PROGRAM main
VAR
	MainGreen : bool := True;
	MainYellow : bool := False;
	MainRed : bool := False;
	SideGreen : bool := False;
	SideYellow : bool := False;
	SideRed : bool := True;
	CarWaiting : bool := False;
	PedWaiting : bool := False;
	GreenTimer : TON;
	YellowTimer : TON;
	SideGreenTimer : TON;
	SideYellowTimer : TON;
	SideYeIIowTimer : dint;
	CycIeActive : bool := False;
	CycleActive : bool := False;
	TON0 : TON;
END_VAR

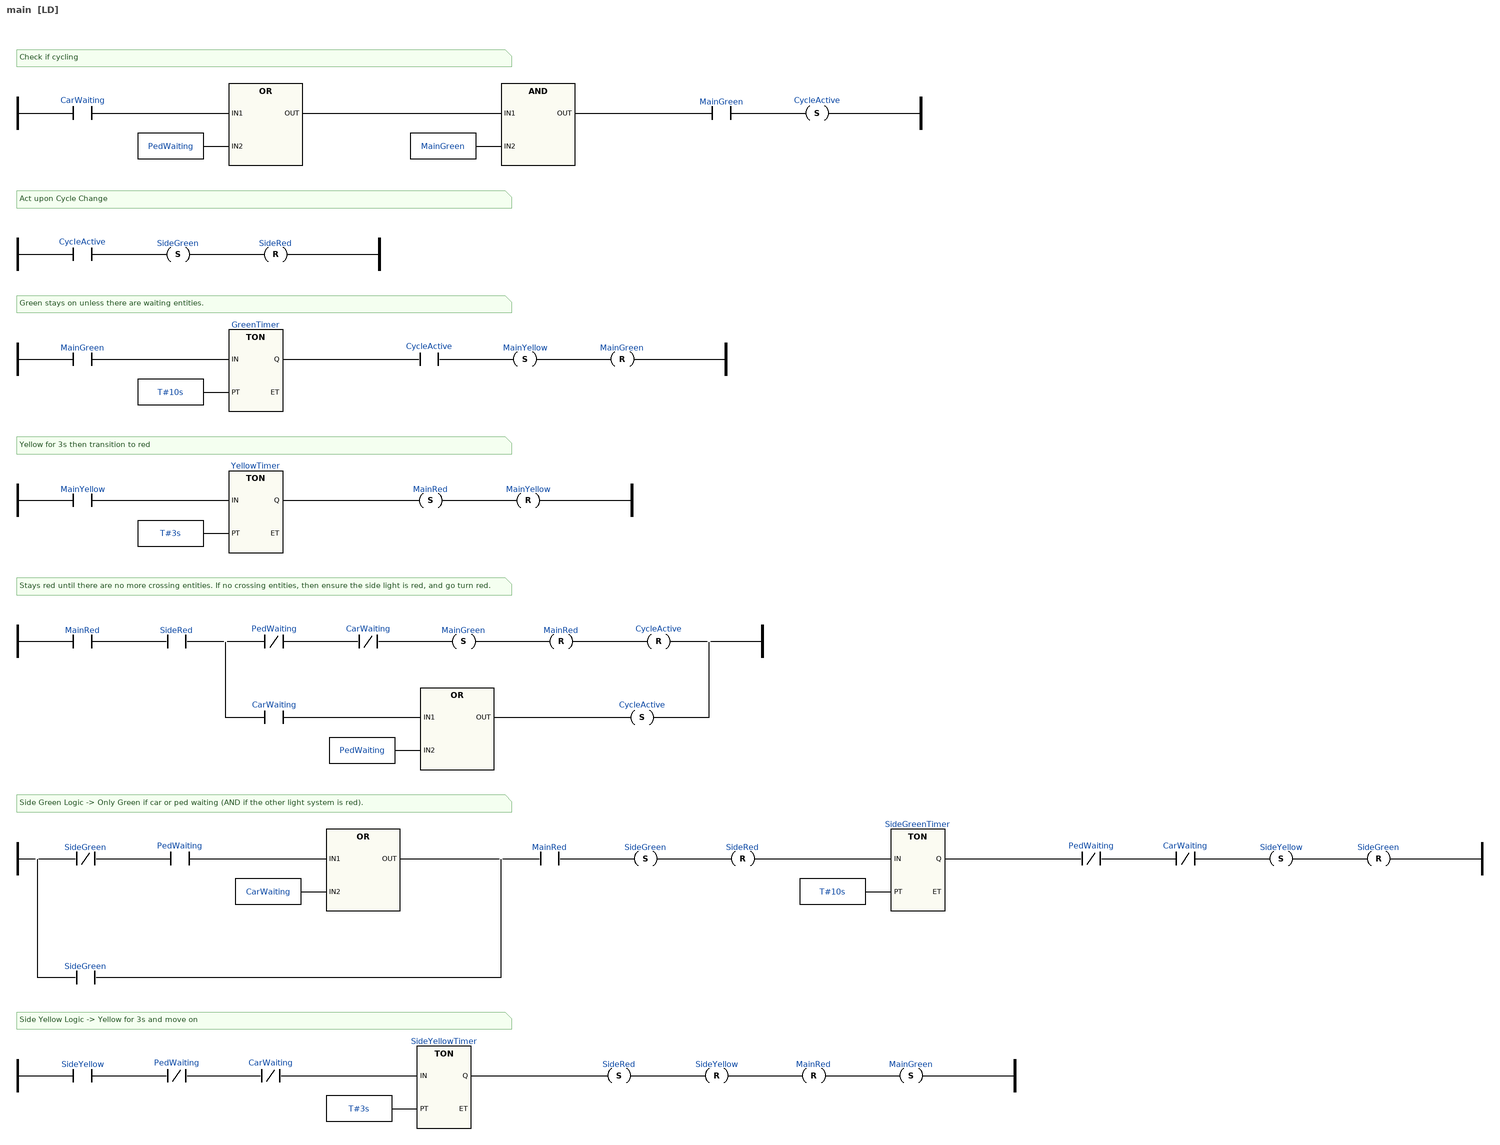
(* LD diagram, written out as Structured Text *)
(* Check if cycling *)
IF (CarWaiting OR PedWaiting) AND MainGreen AND MainGreen THEN CycleActive := TRUE; END_IF;
(* Act upon Cycle Change *)
IF CycIeActive THEN SideGreen := TRUE; END_IF;
IF CycIeActive THEN SideRed := FALSE; END_IF;
(* Green stays on unless there are waiting entities. *)
GreenTimer(IN := MainGreen, PT := T#10s);
IF GreenTimer.Q AND CycleActive THEN MainYellow := TRUE; END_IF;
IF GreenTimer.Q AND CycleActive THEN MainGreen := FALSE; END_IF;
(* Yellow for 3s then transition to red *)
YellowTimer(IN := MainYellow, PT := T#3s);
IF YellowTimer.Q THEN MainRed := TRUE; END_IF;
IF YellowTimer.Q THEN MainYellow := FALSE; END_IF;
(* Stays red until there are no more crossing entities. If no crossing entities, then ensure the side light is red, and go turn red. *)
IF MainRed AND SideRed AND NOT PedWaiting AND NOT CarWaiting THEN MainGreen := TRUE; END_IF;
IF MainRed AND SideRed AND NOT PedWaiting AND NOT CarWaiting THEN MainRed := FALSE; END_IF;
IF MainRed AND SideRed AND NOT PedWaiting AND NOT CarWaiting THEN CycleActive := FALSE; END_IF;
IF MainRed AND SideRed AND CarWaiting OR PedWaiting THEN CycleActive := TRUE; END_IF;
(* Side Green Logic -> Only Green if car or ped waiting (AND if the other light system is red). *)
IF (SideGreen OR NOT SideGreen AND PedWaiting OR CarWaiting) AND MainRed THEN SideGreen := TRUE; END_IF;
IF (SideGreen OR NOT SideGreen AND PedWaiting OR CarWaiting) AND MainRed THEN SideRed := FALSE; END_IF;
SideGreenTimer(IN := (SideGreen OR NOT SideGreen AND PedWaiting OR CarWaiting) AND MainRed, PT := T#10s);
IF SideGreenTimer.Q AND NOT PedWaiting AND NOT CarWaiting THEN SideYellow := TRUE; END_IF;
IF SideGreenTimer.Q AND NOT PedWaiting AND NOT CarWaiting THEN SideGreen := FALSE; END_IF;
(* Side Yellow Logic -> Yellow for 3s and move on *)
SideYellowTimer(IN := SideYellow AND NOT PedWaiting AND NOT CarWaiting, PT := T#3s);
IF SideYellowTimer.Q THEN SideRed := TRUE; END_IF;
IF SideYellowTimer.Q THEN SideYellow := FALSE; END_IF;
IF SideYellowTimer.Q THEN MainRed := FALSE; END_IF;
IF SideYellowTimer.Q THEN MainGreen := TRUE; END_IF;
END_PROGRAM
